	setMessage('Teste Datentyp Array of INT');
	assertEQUAL(s16Value1, s16Value2);
(**********************************************) 	

	u16Value1[0] := 3124;
	u16Value2[0] := 3124;
	
	setMessage('Teste Datentyp UINT');
	assertEQUAL(u16Value1[0] , u16Value2[0] );

	setMessage('Teste Datentyp Array of UINT');
	assertEQUAL(u16Value1 , u16Value2);
(**********************************************) 	

	s32Value1[0] := 1244;
	s32Value2[0] := 1244;
	
	setMessage('Teste Datentyp DINT');
	assertEQUAL(s32Value1[0], s32Value2[0]);

	setMessage('Teste Datentyp Array of DINT');
	assertEQUAL(s32Value1, s32Value2);
(**********************************************) 	

	u32Value1[0] := 4344;
	u32Value2[0] := 4344;
	
	setMessage('Teste Datentyp UDINT');
	assertEQUAL(u32Value1[0], u32Value2[0]);

	setMessage('Teste Datentyp Array of UDINT');
	assertEQUAL(u32Value1, u32Value2);
(**********************************************) 	

	r32Value1[0] := 133.53245;
	r32Value2[0] := 133.53245;
	
	setMessage('Teste Datentyp REAL');
	assertEQUAL(r32Value1[0], r32Value2[0]);

	setMessage('Teste Datentyp Array of REAL');
	assertEQUAL(r32Value1, r32Value2);
(**********************************************) 	

	r64Value1[0] := 1232.53325;
	r64Value2[0] := 1232.53325;

	setMessage('Teste Datentyp LREAL');
	assertEQUAL(r64Value1[0], r64Value2[0]);

	setMessage('Teste Datentyp Array of LREAL');
	assertEQUAL(r64Value1, r64Value2);

(**********************************************) 	

	strValue1[0] := 'Hallo Welt';
	strValue2[0] := 'Hallo Welt';

	setMessage('Teste Datentyp String ist gleich');
	assertStringEqual(ADR(strValue1[0]), ADR(strValue2[0]));

	//setMessage('Teste Datentyp Array of String ist gleich');
	//assertEQUAL(strValue1, strValue2);

	strValue1[0] := 'Hallo Well';
	strValue2[0] := 'Hallo Welt';
	
	setMessage('Teste Datentyp String ist ungleich');
	assertStringNotEqual(ADR(strValue1[0]), ADR(strValue2[0]));

	//setMessage('Teste Datentyp Array of String ist ungleich');
	//assertNotEQUAL(strValue1, strValue2);
	
(**********************************************) 	





	execute := ERetCode_t.eRetDone;
END_METHOD

(******************************************************************************
Baustein: FB_Test_Base.prepare
Spezifikation: doc/Spezifikation.pdf, Kap. x.y.z
-------------------------------------------------------------------------------
erstellt:
von:
Geändert:
von:
-------------------------------------------------------------------------------
Beschreibung
Diese Methode...

-------------------------------------------------------------------------------
Input
-

Output
-
******************************************************************************)
METHOD PUBLIC prepare : ERetCode_t
VAR_INPUT
END_VAR

	prepare := ERetCode_t.eRetDone;
END_METHOD

END_FUNCTION_BLOCK

// ---- Test/FB_Test_Base_Ptr.TcPOU
{attribute 'hide'}
FUNCTION_BLOCK FB_Test_Base_Ptr EXTENDS FB_TestBase
VAR_INPUT
END_VAR
VAR_OUTPUT
END_VAR
VAR
END_VAR

(******************************************************************************
Baustein: FB_Test_Base.cleanup
Spezifikation: doc/Spezifikation.pdf, Kap. x.y.z
-------------------------------------------------------------------------------
erstellt:
von:
Geändert:
von:
-------------------------------------------------------------------------------
Beschreibung
Diese Methode...

-------------------------------------------------------------------------------
Input
-

Output
-
******************************************************************************)
METHOD PUBLIC cleanup : ERetCode_t
VAR_INPUT
END_VAR

	cleanup := ERetCode_t.eRetDone;
END_METHOD

(******************************************************************************
Baustein: FB_Test_Base.execute
Spezifikation: doc/Spezifikation.pdf, Kap. x.y.z
-------------------------------------------------------------------------------
erstellt:
von:
Geändert:
von:
-------------------------------------------------------------------------------
Beschreibung
Diese Methode...

-------------------------------------------------------------------------------
Input
-

Output
-
******************************************************************************)
METHOD PUBLIC execute : ERetCode_t
VAR_INPUT
END_VAR
VAR
	bValue1   : ARRAY[0..10] OF BOOL;
	bValue2   : ARRAY[0..10] OF BOOL;
	s8Value1  : ARRAY[0..10] OF SINT;
	s8Value2  : ARRAY[0..10] OF SINT;
	u8Value1  : ARRAY[0..10] OF USINT;
	u8Value2  : ARRAY[0..10] OF USINT;	
	s16Value1 : ARRAY[0..10] OF INT;
	s16Value2 : ARRAY[0..10] OF INT;
	u16Value1 : ARRAY[0..10] OF UINT;
	u16Value2 : ARRAY[0..10] OF UINT;		
	s32Value1 : ARRAY[0..10] OF DINT;
	s32Value2 : ARRAY[0..10] OF DINT;
	u32Value1 : ARRAY[0..10] OF UDINT;
	u32Value2 : ARRAY[0..10] OF UDINT;	
	r32Value1 : ARRAY[0..10] OF REAL;
	r32Value2 : ARRAY[0..10] OF REAL;
	r64Value1 : ARRAY[0..10] OF LREAL;
	r64Value2 : ARRAY[0..10] OF LREAL;
END_VAR


	bValue1[0] := TRUE;
	bValue2[0] := TRUE;
	
	setMessage('Teste Pointer to BOOL equal');
	assertPtrEQUAL(ADR(bValue1[0]), ADR(bValue1[0]));
	
	setMessage('Teste Pointer to BOOL NOT equal');
	assertPtrNOTEQUAL(ADR(bValue1), ADR(bValue2));

(**********************************************) 
	
	s8Value1[0] := 32;
	s8Value2[0] := 32;
	
	setMessage('Teste Pointer to BOOL SINT equal');
	assertPtrEQUAL(ADR(s8Value1[0]), ADR(s8Value1[0]));

	setMessage('Teste Pointer to SINT not equal');
	assertPtrNOTEQUAL(ADR(s8Value1), ADR(s8Value2));
(**********************************************) 	

	u8Value1[0] := 34;
	u8Value2[0] := 34;
	
	setMessage('Teste Pointer to USINT equal');
	assertPtrEQUAL(ADR(u8Value1[0]), ADR(u8Value1[0]));

	setMessage('Teste Pointer to USINT not equal');
	assertPtrNOTEQUAL(ADR(u8Value1), ADR(u8Value2));
(**********************************************) 	
	
	s16Value1[0] := 1323;
	s16Value2[0] := 1323;
	
	setMessage('Teste Pointer to INT equal');
	assertPtrEQUAL(ADR(s16Value1[0]), ADR(s16Value1[0]));

	setMessage('Teste Pointer to INT not equal');
	assertPtrNOTEQUAL(ADR(s16Value1), ADR(s16Value2));
(**********************************************) 	

	u16Value1[0] := 3124;
	u16Value2[0] := 3124;
	
	setMessage('Teste Pointer to UINT equal');
	assertPtrEQUAL(ADR(u16Value1[0]) , ADR(u16Value1[0]) );

	setMessage('Teste Pointer to  UINT not equal');
	assertPtrNOTEQUAL(ADR(u16Value1) , ADR(u16Value2));
(**********************************************) 	

	s32Value1[0] := 1244;
	s32Value2[0] := 1244;
	
	setMessage('Teste Pointer to DINT equal');
	assertPtrEQUAL(ADR(s32Value1[0]), ADR(s32Value1[0]));

	setMessage('Teste Pointer to  DINT not equal');
	assertPtrNOTEQUAL(ADR(s32Value1), ADR(s32Value2));
(**********************************************) 	

	u32Value1[0] := 4344;
	u32Value2[0] := 4344;
	
	setMessage('Teste Pointer to UDINT equal');
	assertPtrEQUAL(ADR(u32Value1[0]), ADR(u32Value1[0]));

	setMessage('Teste Pointer to  UDINT not equal');
	assertPtrNOTEQUAL(ADR(u32Value1), ADR(u32Value2));
(**********************************************) 	

	r32Value1[0] := 133.53245;
	r32Value2[0] := 133.53245;
	
	setMessage('Teste Pointer to REAL equal');
	assertPtrEQUAL(ADR(r32Value1[0]), ADR(r32Value1[0]));

	setMessage('Teste Pointer to  REAL not equal');
	assertPtrNOTEQUAL(ADR(r32Value1), ADR(r32Value2));
(**********************************************) 	

	r64Value1[0] := 1232.53325;
	r64Value2[0] := 1232.53325;

	setMessage('Teste Pointer to LREAL equal');
	assertPtrEQUAL(ADR(r64Value1[0]), ADR(r64Value1[0]));

	setMessage('Teste Pointer to LREAL not equal');
	assertPtrNOTEQUAL(ADR(r64Value1), ADR(r64Value2));

(**********************************************)

	setMessage('Teste Pointer = 0');	
	assertPtrNull(pActual := 0);
	
	setMessage('Teste Pointer <> 0');	
	assertPtrNotNull(pActual := ADR(r32Value1[0]));	
	
(**********************************************)	
	
	
	
	
	
	
	
	
	
	execute := ERetCode_t.eRetDone;
END_METHOD

(******************************************************************************
Baustein: FB_Test_Base.prepare
Spezifikation: doc/Spezifikation.pdf, Kap. x.y.z
-------------------------------------------------------------------------------
erstellt:
von:
Geändert:
von:
-------------------------------------------------------------------------------
Beschreibung
Diese Methode...

-------------------------------------------------------------------------------
Input
-

Output
-
******************************************************************************)
METHOD PUBLIC prepare : ERetCode_t
VAR_INPUT
END_VAR

	prepare := ERetCode_t.eRetDone;
END_METHOD

END_FUNCTION_BLOCK

// ---- Test/FB_Test_Base_Not.TcPOU
{attribute 'hide'}
FUNCTION_BLOCK FB_Test_Base_Not EXTENDS FB_TestBase
VAR_INPUT
END_VAR
VAR_OUTPUT
END_VAR
VAR
END_VAR

(******************************************************************************
Baustein: FB_Test_Base_Not.cleanup
Spezifikation: doc/Spezifikation.pdf, Kap. x.y.z
-------------------------------------------------------------------------------
erstellt:
von:
Geändert:
von:
-------------------------------------------------------------------------------
Beschreibung
Diese Methode...

-------------------------------------------------------------------------------
Input
-

Output
-
******************************************************************************)
METHOD PUBLIC cleanup : ERetCode_t
VAR_INPUT
END_VAR

	cleanup := ERetCode_t.eRetDone;
END_METHOD

(******************************************************************************
Baustein: FB_Test_Base_Not.execute
Spezifikation: doc/Spezifikation.pdf, Kap. x.y.z
-------------------------------------------------------------------------------
erstellt:
von:
Geändert:
von:
-------------------------------------------------------------------------------
Beschreibung
Diese Methode...

-------------------------------------------------------------------------------
Input
-

Output
-
******************************************************************************)
METHOD PUBLIC execute : ERetCode_t
VAR_INPUT
END_VAR
VAR
	bValue1   : ARRAY[0..10] OF BOOL;
	bValue2   : ARRAY[0..10] OF BOOL;
	s8Value1  : ARRAY[0..10] OF SINT;
	s8Value2  : ARRAY[0..10] OF SINT;
	u8Value1  : ARRAY[0..10] OF USINT;
	u8Value2  : ARRAY[0..10] OF USINT;	
	s16Value1 : ARRAY[0..10] OF INT;
	s16Value2 : ARRAY[0..10] OF INT;
	u16Value1 : ARRAY[0..10] OF UINT;
	u16Value2 : ARRAY[0..10] OF UINT;		
	s32Value1 : ARRAY[0..10] OF DINT;
	s32Value2 : ARRAY[0..10] OF DINT;
	u32Value1 : ARRAY[0..10] OF UDINT;
	u32Value2 : ARRAY[0..10] OF UDINT;	
	r32Value1 : ARRAY[0..10] OF REAL;
	r32Value2 : ARRAY[0..10] OF REAL;
	r64Value1 : ARRAY[0..10] OF LREAL;
	r64Value2 : ARRAY[0..10] OF LREAL;
END_VAR


	bValue1[0] := FALSE;
	bValue2[0] := TRUE;
	
	setMessage('Teste Datentyp BOOL');
	assert.NotEQUAL(bValue1[0], bValue2[0]);
	
	setMessage('Teste Datentyp Array of BOOL');
	assert.NotEQUAL(bValue1, bValue2);

(**********************************************) 
	
	s8Value1[0] := 31;
	s8Value2[0] := 32;
	
	setMessage('Teste Datentyp SINT');
	assert.NotEQUAL(s8Value1[0], s8Value2[0]);

	setMessage('Teste Datentyp Array SINT');
	assert.NotEQUAL(s8Value1, s8Value2);
(**********************************************) 	

	u8Value1[0] := 1;
	u8Value2[0] := 34;
	
	setMessage('Teste Datentyp USINT');
	assert.NotEQUAL(u8Value1[0], u8Value2[0]);

	setMessage('Teste Datentyp Array of USINT');
	assert.NotEQUAL(u8Value1, u8Value2);
(**********************************************) 	
	
	s16Value1[0] := 1323;
	s16Value2[0] := 4324;
	
	setMessage('Teste Datentyp INT');
	assert.NotEQUAL(s16Value1[0], s16Value2[0]);

	setMessage('Teste Datentyp Array of INT');
	assert.NotEQUAL(s16Value1, s16Value2);
(**********************************************) 	

	u16Value1[0] := 3124;
	u16Value2[0] := 4232;
	
	setMessage('Teste Datentyp UINT');
	assert.NotEQUAL(u16Value1[0] , u16Value2[0] );

	setMessage('Teste Datentyp Array of UINT');
	assert.NotEQUAL(u16Value1 , u16Value2);
(**********************************************) 	

	s32Value1[0] := 1244;
	s32Value2[0] := 1593;
	
	setMessage('Teste Datentyp DINT');
	assert.NotEQUAL(s32Value1[0], s32Value2[0]);

	setMessage('Teste Datentyp Array of DINT');
	assert.NotEQUAL(s32Value1, s32Value2);
(**********************************************) 	

	u32Value1[0] := 4344;
	u32Value2[0] := 3424;
	
	setMessage('Teste Datentyp UDINT');
	assert.NotEQUAL(u32Value1[0], u32Value2[0]);

	setMessage('Teste Datentyp Array of UDINT');
	assert.NotEQUAL(u32Value1, u32Value2);
(**********************************************) 	

	r32Value1[0] := 133.53245;
	r32Value2[0] := 5345.53245;
	
	setMessage('Teste Datentyp REAL');
	assert.NotEQUAL(r32Value1[0], r32Value2[0]);

	setMessage('Teste Datentyp Array of REAL');
	assert.NotEQUAL(r32Value1, r32Value2);
(**********************************************) 	

	r64Value1[0] := 1232.53325;
	r64Value2[0] := 1345.53325;

	setMessage('Teste Datentyp LREAL');
	assert.NotEQUAL(r64Value1[0], r64Value2[0]);

	setMessage('Teste Datentyp Array of LREAL');
	assert.NotEQUAL(r64Value1, r64Value2);

(**********************************************) 		
	execute := ERetCode_t.eRetDone;
END_METHOD

(******************************************************************************
Baustein: FB_Test_Base_Not.prepare
Spezifikation: doc/Spezifikation.pdf, Kap. x.y.z
-------------------------------------------------------------------------------
erstellt:
von:
Geändert:
von:
-------------------------------------------------------------------------------
Beschreibung
Diese Methode...

-------------------------------------------------------------------------------
Input
-

Output
-
******************************************************************************)
METHOD PUBLIC prepare : ERetCode_t
VAR_INPUT
END_VAR

	prepare := ERetCode_t.eRetDone;
END_METHOD

END_FUNCTION_BLOCK

// ---- Test/FB_Test_Base_Delay.TcPOU
{attribute 'hide'}
FUNCTION_BLOCK FB_Test_Base_Delay EXTENDS FB_TestBase
VAR_INPUT
END_VAR
VAR_OUTPUT
END_VAR
VAR
	fbDelay : TON;
END_VAR

(******************************************************************************
Baustein: FB_Test_Base_Delay.cleanup
Spezifikation: doc/Spezifikation.pdf, Kap. x.y.z
-------------------------------------------------------------------------------
erstellt:
von:
Geändert:
von:
-------------------------------------------------------------------------------
Beschreibung
Diese Methode...

-------------------------------------------------------------------------------
Input
-

Output
-
******************************************************************************)
METHOD PUBLIC cleanup : ERetCode_t
VAR_INPUT
END_VAR

	cleanup := ERetCode_t.eRetDone;
	
	fbDelay(IN := false);
END_METHOD

(******************************************************************************
Baustein: FB_Test_Base_Delay.execute
Spezifikation: doc/Spezifikation.pdf, Kap. x.y.z
-------------------------------------------------------------------------------
erstellt:
von:
Geändert:
von:
-------------------------------------------------------------------------------
Beschreibung
Diese Methode...

-------------------------------------------------------------------------------
Input
-

Output
-
******************************************************************************)
METHOD PUBLIC execute : ERetCode_t
VAR_INPUT
END_VAR
VAR
	bValue1  : BOOL;
	bValue2  : BOOL;
	s32Value1 : DINT;
	s32Value2 : DINT;
	r32Value1 : REAL;
	r32Value2 : REAL;
END_VAR

	fbDelay(PT := t#250ms);
	execute 	  := ERetCode_t.eRetBusy;

	bValue1 := TRUE;
	bValue2 := TRUE;
	assertEQUAL(bValue1, bValue2);

	s32Value1 := 1593;
	s32Value2 := 1593;
	assertEQUAL(s32Value1, s32Value2);

	r32Value1 := 5345.53245;
	r32Value2 := 5345.53245;
	assertEQUAL(r32Value1, r32Value2);

	if fbDelay.Q then
		execute := ERetCode_t.eRetDone;
	end_if;
END_METHOD

(******************************************************************************
Baustein: FB_Test_Base_Delay.prepare
Spezifikation: doc/Spezifikation.pdf, Kap. x.y.z
-------------------------------------------------------------------------------
erstellt:
von:
Geändert:
von:
-------------------------------------------------------------------------------
Beschreibung
Diese Methode...

-------------------------------------------------------------------------------
Input
-

Output
-
******************************************************************************)
METHOD PUBLIC prepare : ERetCode_t
VAR_INPUT
END_VAR

	prepare := ERetCode_t.eRetDone;
	
	fbDelay.IN := true;
END_METHOD

END_FUNCTION_BLOCK
